PROGRAM P60_UpdatePV
VAR
	i: UINT;
END_VAR

FOR i:=1 TO GVL_IO.NumFlowController DO
	GVL_IO.aController_PV[i] := (INT_TO_REAL(GVL_IO.aAnalogInputIO[i]) / GVL_IO.KL3464MaxValueH) * GVL_IO.AnalogControllerOutputVoltage;
END_FOR

GVL_IO.aController_PV[27] := WORD_TO_REAL(GVL_IO.wE3508_PV);
GVL_IO.aController_PV[28] := WORD_TO_REAL(GVL_IO.wIqPlus_CDG2_PV);
GVL_IO.aController_PV[29] := GVL_IO.nRotation_Converted_PV;

END_PROGRAM

(* stored: Version 1.1.0.1, ProductVersion 3.1.4026.11
   POU P60_UpdatePV: Id {f8956921-3779-4dbc-8078-a6d7c5df8142}, SpecialFunc None *)
